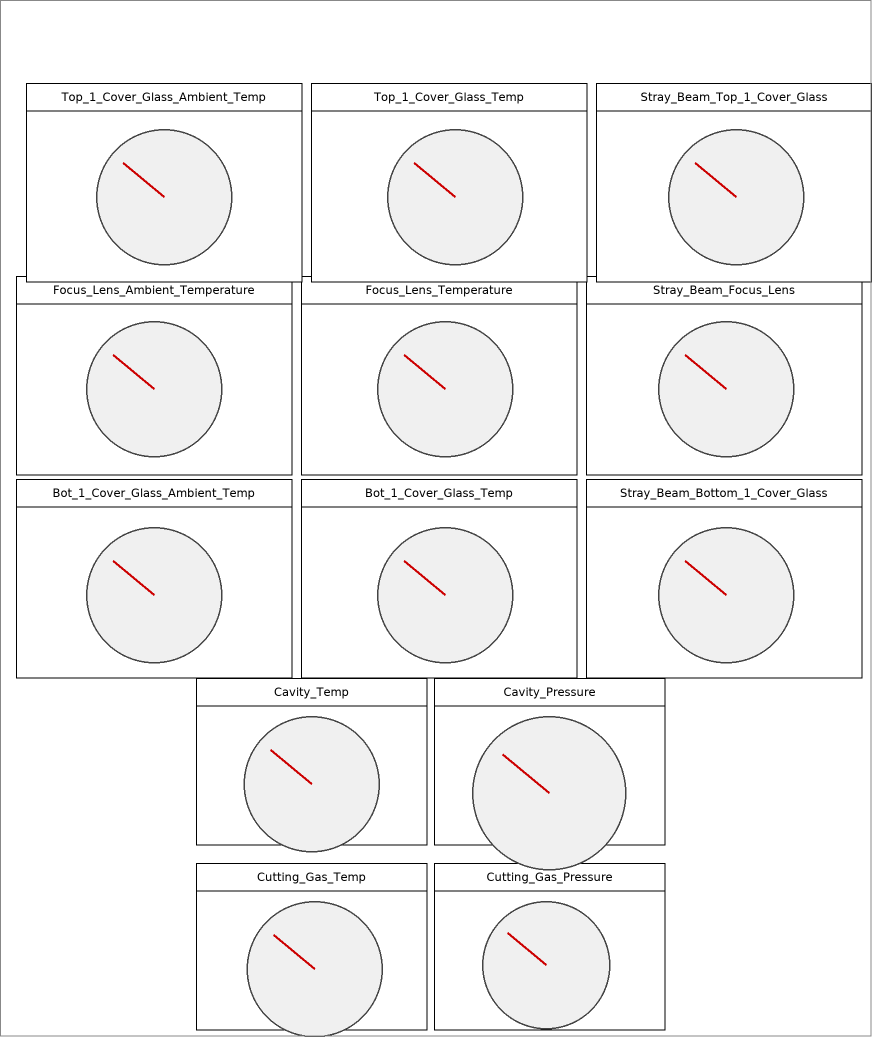
VISUALIZATION Visualization_1  // 872x1037
    Rectangle (196,678 231x167)
    Rectangle (196,678 231x28), "Cavity_Temp"
    Rectangle (196,863 231x167)
    Rectangle (196,863 231x28), "Cutting_Gas_Temp"
    Rectangle (434,678 231x167)
    Rectangle (434,678 231x28), "Cavity_Pressure"
    Rectangle (434,863 231x167)
    Rectangle (434,863 231x28), "Cutting_Gas_Pressure"
    Meter180 (199,716 225x136), value: Data11_Cavity_Temp/100, style: Meter-Meter180-Blue, scale format: %.1f, scale 0..60
        p518627256: °C
    Meter180 (202,901 225x136), value: Data13_Cutting_Gas_Temp/100, style: Meter-Meter180-Blue, scale format: %.1f, scale 0..60
        p518627256: °C
    Meter180 (437,716 224x154), value: Data12_Cavity_Pressure/10, style: Meter-Meter180-Blue, scale format: %.1f, scale 0..10
        p518627256: Bars
    Meter180 (434,901 224x128), value: Data14_Cutting_Gas_Pressure/10, style: Meter-Meter180-Blue, scale format: %.1f, scale 0..10
        p518627256: Bars
    Rectangle (586,479 276x199)
    Rectangle (586,276 276x199)
    Rectangle (301,479 276x199)
    Rectangle (301,276 276x199)
    Rectangle (16,276 276x199)
    Rectangle (16,479 276x199)
    Rectangle (16,276 276x28), "Focus_Lens_Ambient_Temperature"
    Rectangle (301,276 276x28), "Focus_Lens_Temperature"
    Rectangle (16,479 276x28), "Bot_1_Cover_Glass_Ambient_Temp"
    Rectangle (301,479 276x28), "Bot_1_Cover_Glass_Temp"
    Rectangle (586,276 276x28), "Stray_Beam_Focus_Lens"
    Rectangle (586,479 276x28), "Stray_Beam_Bottom_1_Cover_Glass"
    Meter180 (29,321 250x136), value: Data03_Focus_Lens_Ambient_Temperature/100, style: Meter-Meter180-Gray, scale format: %.1f, scale 0..30
        p518627256: °C
    Meter180 (29,527 250x136), value: Data09_Bottom_1_Cover_Glass_Ambient_Temp/100, style: Meter-Meter180-Gray, scale format: %.1f, scale 0..30
        p518627256: °C
    Meter180 (320,321 250x136), value: Data04_Focus_Lens_Temperature/100, style: Meter-Meter180-Gray, scale format: %.1f, scale 0..60
        p518627256: °C
    Meter180 (320,527 250x136), value: Data10_Bottom_1_Cover_Glasst_Temp/100, style: Meter-Meter180-Gray, scale format: %.1f, scale 0..60
        p518627256: °C
    Meter180 (601,321 250x136), value: Data28_Stray_Beam_Focus_Lens/100, style: Meter-Meter180-Gray, scale format: %.1f, scale 0..30
        p518627256: °C
    Meter180 (601,527 250x136), value: Data29_Stray_Beam_Bottom_1_Cover_Glass/100, style: Meter-Meter180-Gray, scale format: %.1f, scale 0..30
        p518627256: °C
    Rectangle (596,83 276x199)
    Rectangle (311,83 276x199)
    Rectangle (26,83 276x199)
    Rectangle (26,83 276x28), "Top_1_Cover_Glass_Ambient_Temp"
    Rectangle (311,83 276x28), "Top_1_Cover_Glass_Temp"
    Rectangle (596,83 276x28), "Stray_Beam_Top_1_Cover_Glass"
    Meter180 (39,129 250x136), value: Data07_Top_1_Cover_Glass_Ambient_Temp/100, style: Meter-Meter180-Gray, scale format: %.1f, scale 0..30
        p518627256: °C
    Meter180 (330,129 250x136), value: Data08_Top_1_Cover_Glass_Temp/100, style: Meter-Meter180-Gray, scale format: %.1f, scale 0..60
        p518627256: °C
    Meter180 (611,129 250x136), value: Data27_Stray_Beam_Top_1_Cover_Glass/100, style: Meter-Meter180-Gray, scale format: %.1f, scale 0..30
        p518627256: °C
END_VISUALIZATION

(* stored: Version 1.1.0.1
   Visu Visualization_1: Id {61de5836-1d24-4e5b-9a3f-137ea7dbc579} *)
